// SIMATIC S7-200 project (STEP 7-Micro/WIN), CPU 224 REL 01.22

ORGANIZATION_BLOCK MAIN:OB1
TITLE=PROGRAM COMMENTS
BEGIN
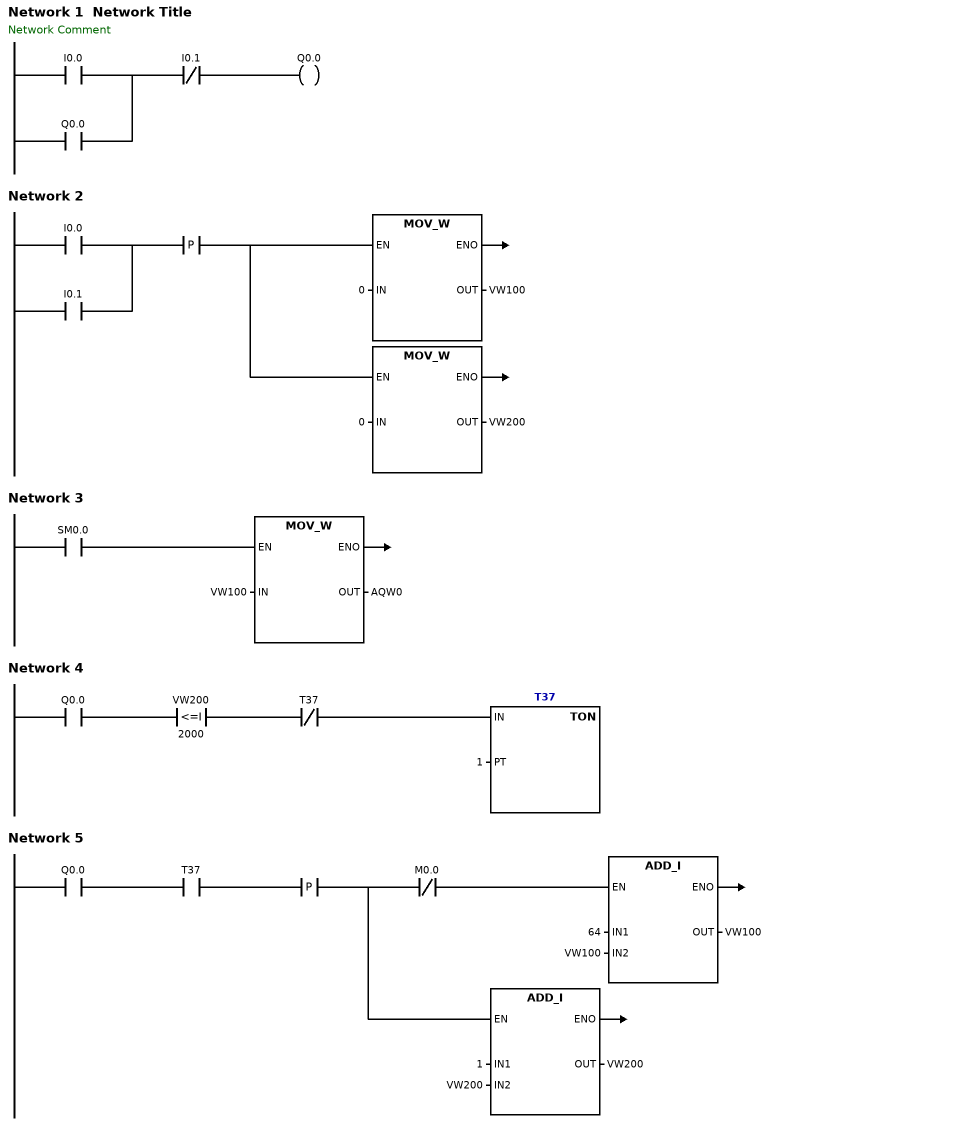
Network 1 // Network Title
// Network Comment
LD     I0.0
O      Q0.0
AN     I0.1
=      Q0.0
Network 2
LD     I0.0
O      I0.1
EU
MOVW   0, VW100
MOVW   0, VW200
Network 3
LD     SM0.0
MOVW   VW100, AQW0
Network 4
LD     Q0.0
AW<=   VW200, 2000
AN     T37
TON    T37, 1
Network 5
LD     Q0.0
A      T37
EU
LPS
AN     M0.0
+I     64, VW100
LPP
+I     1, VW200
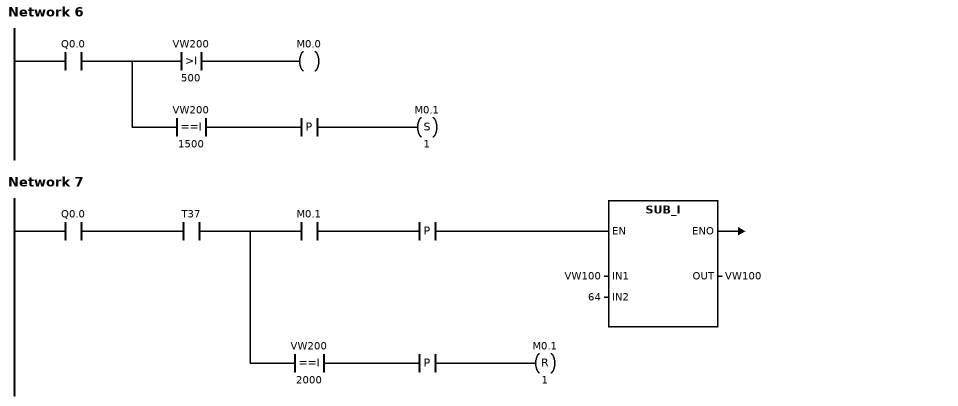
Network 6
LD     Q0.0
LPS
AW>    VW200, 500
=      M0.0
LPP
AW=    VW200, 1500
EU
S      M0.1, 1
Network 7
LD     Q0.0
A      T37
LPS
A      M0.1
EU
-I     64, VW100
LPP
AW=    VW200, 2000
EU
R      M0.1, 1
END_ORGANIZATION_BLOCK
